FUNCTION_BLOCK I_VDS (* Vehicle Direction/Speed VDS *)
  (* Standard: ISO 11783-7; Classification: PGN 65256; Function: Vehicle Direction/Speed VDS; Description: Copyright (c) 2024 HR Agrartechnik GmbH This program and the accompanying materials are made available under the terms of the Eclipse Public License 2.0 which is available at https://www.eclipse.org/legal/epl-2.0/ SPDX-License-Identifier: EPL-2.0 See https://copperhilltech.com/sae-j1939-gps-module/ for details https://docs.ms-muc-docs.de/projects/isobus-other-docs/de/latest/PGN/PGN_65256.html *)
  (* Version 1.0, 2024-07-09, Franz Hoepfinger, HR Agrartechnik GmbH *)
  PACKAGE isobus::tecu;
  IMPORT eclipse4diac::core::TypeHash;
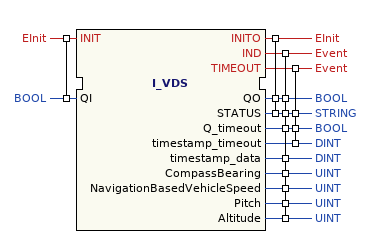
  EVENT_INPUT
    INIT : EInit WITH QI; (* Service Initialization *)
  END_EVENT
  EVENT_OUTPUT
    INITO : EInit WITH QO, STATUS; (* Initialization Confirm *)
    IND WITH QO, timestamp_data, CompassBearing, NavigationBasedVehicleSpeed, Pitch, STATUS, Q_timeout, Altitude; (* Indication from Resource *)
    TIMEOUT WITH timestamp_timeout, STATUS, Q_timeout;
  END_EVENT
  VAR_INPUT
    QI : BOOL; (* Event Input Qualifier *)
  END_VAR
  VAR_OUTPUT
    QO : BOOL; (* Event Output Qualifier *)
    STATUS : STRING;
    Q_timeout : BOOL;
    timestamp_timeout : DINT;
    timestamp_data : DINT;
    CompassBearing : UINT; (* Present compass bearing of vehicle. *) {SET_ATTRIBUTE(SPN, 165)} {SET_ATTRIBUTE(SP_Name, 'Compass Bearing')} {SET_ATTRIBUTE(SP_Position_In_PG, '1')} {SET_ATTRIBUTE(SP_Length, 2)} (* 2 bytes *) {SET_ATTRIBUTE(Scaling, '1/128 deg per bit')} {SET_ATTRIBUTE(Offset, )} {SET_ATTRIBUTE(Link, 'https://docs.ms-muc-docs.de/projects/isobus-other-docs/de/latest/PGN/PGN_65256.html#spn-165-compassbearing-kompassrichtung')}
    NavigationBasedVehicleSpeed : UINT; (* Speed of the vehicle as calculated from a device such as a Global Positioning System (GPS). *) {SET_ATTRIBUTE(SPN, 517)} {SET_ATTRIBUTE(SP_Name, 'Navigation-Based Vehicle Speed')} {SET_ATTRIBUTE(SP_Position_In_PG, '2')} {SET_ATTRIBUTE(SP_Length, 2)} (* 2 bytes *) {SET_ATTRIBUTE(Scaling, '1/256 km/h per bit')} {SET_ATTRIBUTE(Offset, )} {SET_ATTRIBUTE(Link, 'https://docs.ms-muc-docs.de/projects/isobus-other-docs/de/latest/PGN/PGN_65256.html#spn-517-navigationbasedvehiclespeed-fahrzeuggeschwindigkeit')}
    Pitch : UINT; (* Pitch (rotation about the y-axis) of the vehicle as calculated by the navigation device(s). *) {SET_ATTRIBUTE(SPN, 583)} {SET_ATTRIBUTE(SP_Name, 'Pitch')} {SET_ATTRIBUTE(SP_Position_In_PG, '3')} {SET_ATTRIBUTE(SP_Length, 2)} (* 2 bytes *) {SET_ATTRIBUTE(Scaling, 'Not used; Always set to 0xFFFF')} {SET_ATTRIBUTE(Offset, )} {SET_ATTRIBUTE(Link, 'https://docs.ms-muc-docs.de/projects/isobus-other-docs/de/latest/PGN/PGN_65256.html#spn-583-pitch-neigungswinkel')}
    Altitude : UINT; (* Altitude of the vehicle referenced to sea level at standard atmospheric pressure and temperature. *) {SET_ATTRIBUTE(SPN, 580)} {SET_ATTRIBUTE(SP_Name, 'Altitude')} {SET_ATTRIBUTE(SP_Position_In_PG, '4')} {SET_ATTRIBUTE(SP_Length, 2)} (* 2 bytes *) {SET_ATTRIBUTE(Scaling, 'Not used; Always set to 0xFFFF')} {SET_ATTRIBUTE(Offset, )} {SET_ATTRIBUTE(Link, 'https://docs.ms-muc-docs.de/projects/isobus-other-docs/de/latest/PGN/PGN_65256.html#spn-580-altitude-hohe-uber-dem-meeresspiegel')}
  END_VAR
END_FUNCTION_BLOCK
